// TIA Portal project "FactoryIO_Template_S7-1200_V15_V15.1" (V15.1)
// Vorlageprojekt für das Buch mit Zielsystem S7-1200

(* hardware
DEVICE "S7-1200-Station_1"  S7-1200 Station
   slot 0: "Baugruppenträger_0"  Rack  V1.0
   slot 1: "PLC_1"  CPU 1211C DC/DC/DC  6ES7 211-1AE40-0XB0  V4.1
DEVICE "HMI_1"  KTP900 Basic PN
   slot 0: "HMI_1"  KTP900 Basic PN  6AV2 123-2JB03-0AX0  15.1.0.0
   slot 1: "HMI_RT_1"  KTP900 Basic PN  6AV2 123-2JB03-0AX0  15.1.0.0
   slot 5: "HMI_1.IE_CP_1"  PROFINET Interface  15.0.1.0
      slot 1: "PROFINET Interface_1"  PROFINET Interface
         slot 1: "Port_1"  Port
*)

// ===== PLC "PLC_1"  CPU 1211C DC/DC/DC =====

VAR_GLOBAL   // PLC tag table "Standard-Variablentabelle"
   "Fill valve" AT %A0.0 : Bool;
   "Fill" AT %E0.0 : Bool;
   "Discharge" AT %E0.1 : Bool;
   "Filling" AT %Q0.1 : Bool;
   "Discharge valve" AT %Q0.2 : Bool;
   "Discharging" AT %Q0.3 : Bool;
   "Timer" AT %QD30 : DInt;
   "reset_fill" AT %I0.3 : Bool;
   "reset_empty" AT %I0.4 : Bool;
END_VAR

DATA_BLOCK "Auxiliare"   // DB1
{ S7_Optimized_Access := 'TRUE' }
VERSION : 0.1
   VAR
      timp_setat : Time;
      timp_setat_secunde : Time;
      timp_trecut : Time;
      timp_trecut_secunde_DInt : DInt;
   END_VAR
BEGIN
END_DATA_BLOCK

// folder: System blocks/Program resources

DATA_BLOCK "timer_umplere"   // DB2
{ S7_Optimized_Access := 'TRUE' }
AUTHOR : Simatic
FAMILY : IEC
NAME : IEC_TMR
VERSION : 1.0
// stored: InstanceOfName IEC_TIMER
"IEC_TIMER"
BEGIN
END_DATA_BLOCK

// folder: (top level)

FUNCTION "MHJ-PLC-Lab-Function-S71200" : Void   // FC9000, SCL
{ S7_Optimized_Access := 'TRUE' }
VERSION : 0.1
   VAR_TEMP
      rdTimeReturn : Int;
      outputTime : DTL;
      SyncVal : Byte;
      forVal : Int;
      forVal_2 : Int;
      Value : Byte;
   END_VAR
   VAR CONSTANT
      CompVal : Byte := 16#34;
      Value_01 : Byte := 16#11;
      Value_01_DW : DWord := 16#A165_D992;
      Value_02_DW : DWord := 16#58BE_4401;
   END_VAR
BEGIN

   #Value:=PEEK(area := 16#82,
        dbNumber := 0,
        byteOffset := 511);
   #Value := #Value + 1;

   POKE(area := 16#82,
        dbNumber := 0,
        byteOffset := 511,
        value := #Value);

   POKE(area:=16#81,
        dbNumber:=0,
        byteOffset:=1016,
        value:=#Value_01_DW);
   POKE(area := 16#81,
        dbNumber := 0,
        byteOffset := 1020,
        value := #Value_02_DW);

   POKE(area := 16#81,
        dbNumber := 0,
        byteOffset := 511,
        value := B#16#00);

   FOR #forVal := 0 TO 120 DO
       FOR #forVal_2:=0 TO 10 DO
           #rdTimeReturn:=RD_SYS_T(#outputTime);
           #rdTimeReturn := WR_SYS_T(#outputTime);
           #rdTimeReturn := RD_SYS_T(#outputTime);
           #rdTimeReturn := WR_SYS_T(#outputTime);
       END_FOR;
       #SyncVal:= PEEK(area := 16#81,
                      dbNumber := 0,
                      byteOffset := 511);
       IF #SyncVal = #CompVal THEN
          GOTO M_1;
       END_IF;
   END_FOR;
   RETURN;

   M_1:
   POKE(area := 16#81,
        dbNumber := 0,
        byteOffset := 511,
        value := B#16#0);
END_FUNCTION

ORGANIZATION_BLOCK "Main"   // OB1, LAD, ProgramCycle
TITLE = "Main Program Sweep (Cycle)"
{ S7_Optimized_Access := 'TRUE' }
VERSION : 0.1
   VAR_INPUT
      Initial_Call : Bool;   // Initial call of this OB
      Remanence : Bool;   // =True, if remanent data are available
   END_VAR
BEGIN

REGION Network 1: Konnektierungsbaustein für PLC-Lab
   // Im Netzwerk 1 wird der Konnektierungsbaustein für PLC-Lab aufgerufen.
   // Dieser Aufruf darf nicht entfernt werden!
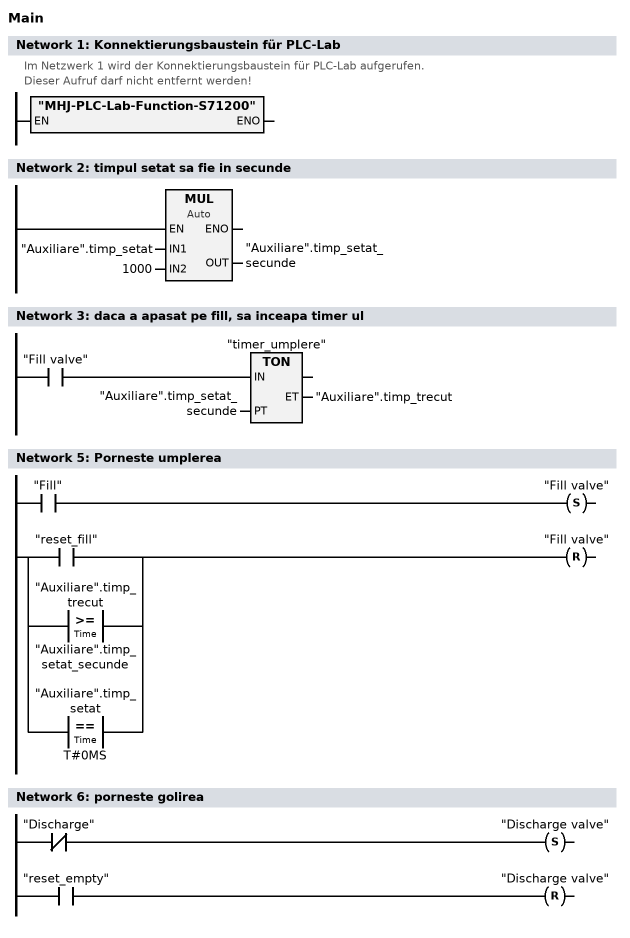
   RUNG wire#powerrail
      "MHJ-PLC-Lab-Function-S71200"()
   END_RUNG
   // the same network as SCL:
   "MHJ-PLC-Lab-Function-S71200"();
END_REGION

REGION Network 2: timpul setat sa fie in secunde
   RUNG wire#powerrail
      Mul(in1 := "Auxiliare".timp_setat, in2 := 1000, out => "Auxiliare".timp_setat_secunde)
   END_RUNG
   // the same network as SCL:
   "Auxiliare".timp_setat_secunde := "Auxiliare".timp_setat * 1000;
END_REGION

REGION Network 3: daca a apasat pe fill, sa inceapa timer ul
   "timer_umplere".TON(IN := "Fill valve", PT := "Auxiliare".timp_setat_secunde, ET => "Auxiliare".timp_trecut);
END_REGION

REGION Network 4 (SCL): timp de afisat in secunde
   "Timer" := TIME_TO_DINT("Auxiliare".timp_trecut / 1000);
END_REGION

REGION Network 5: Porneste umplerea
   RUNG wire#powerrail
      Contact( "Fill" )
      S_Coil( "Fill valve" )
   END_RUNG
   RUNG wire#powerrail
      Contact( "reset_fill" )
      wire#w1
      R_Coil( "Fill valve" )
   END_RUNG
   RUNG wire#powerrail
      { S7_Templates := "SrcType := Time" } GE_Contact(in1 := "Auxiliare".timp_trecut, in2 := "Auxiliare".timp_setat_secunde)
   END_RUNG wire#w1
   RUNG wire#powerrail
      { S7_Templates := "SrcType := Time" } EQ_Contact(in1 := "Auxiliare".timp_setat, in2 := T#0MS)
   END_RUNG wire#w1
   // the same network as SCL:
   IF "Fill" THEN "Fill valve" := TRUE; END_IF;
   IF "reset_fill" OR ("Auxiliare".timp_trecut >= "Auxiliare".timp_setat_secunde) OR ("Auxiliare".timp_setat = T#0MS) THEN
       "Fill valve" := FALSE;
   END_IF;
END_REGION

REGION Network 6: porneste golirea
   RUNG wire#powerrail
      I_Contact( "Discharge" )
      S_Coil( "Discharge valve" )
   END_RUNG
   RUNG wire#powerrail
      Contact( "reset_empty" )
      R_Coil( "Discharge valve" )
   END_RUNG
   // the same network as SCL:
   IF NOT "Discharge" THEN "Discharge valve" := TRUE; END_IF;
   IF "reset_empty" THEN "Discharge valve" := FALSE; END_IF;
END_REGION
END_ORGANIZATION_BLOCK

(* ===== HMI "HMI_RT_1" =====
system functions are stored by id; their names below are inferred from use
connection "HMI_Connection_1": ETHERNET, SMART_S7_1200_OMS

HMI tags "Default tag table"
   "Auxiliare_timp" : Time = PLC Auxiliare.timp_setat, 1 s
   "Auxiliare_timp_trecut_secunde_DInt" : DInt = PLC Auxiliare.timp_trecut_secunde_DInt, 1 s
   "Timer" : DInt = PLC Timer AT %QD30, 1 s
   "Fill" : Bool = PLC Fill AT %I0.0, 1 s
   "Discharge" : Bool = PLC Discharge AT %I0.1, 1 s
   "reset_fill" : Bool = PLC reset_fill AT %I0.3, 1 s
   "reset_empty" : Bool = PLC reset_empty AT %I0.4, 1 s

Template "Template_1" 800x480
   Button "Exit" at 722,440 size 55x39; TextOff 'Exit'; PictureOff "ExitRuntime_KTP900_Basic_PN_TR"; PictureOn "ExitRuntime_KTP900_Basic_PN_TR"
      on Release: StopRuntime(0)
   Button "Template_Button" at 622,440 size 55x39; TextOff 'Text'
   Button "Template_Button_1" at 522,440 size 55x39; TextOff 'Text'
   Button "Template_Button_2" at 422,440 size 55x39; TextOff 'Text'
   Button "Template_Button_3" at 322,440 size 55x39; TextOff 'Text'
   Button "Template_Button_4" at 222,440 size 55x39; TextOff 'Text'
   Button "Template_Button_5" at 122,440 size 55x39; TextOff 'Text'
   Button "Start screen" at 22,440 size 55x39; TextOff 'Start screen'; PictureOff "NavigateHome_KTP900_Basic_PN_TR"; PictureOn "NavigateHome_KTP900_Basic_PN_TR"
      on Release: ActivateScreen("Main", 0)

screen "Main" 800x480, template "Template_1"
   IOField "I/O field_1" at 365,126 size 60x32; FormatPattern 999; Unit s
      ProcessValue <- "Auxiliare_timp"
   TextField "Text field_1" at 357,100 size 74x20; Text 'Timp Setat'
   IOField "I/O field_2" at 366,200 size 59x32; FormatPattern 999; Unit s
      ProcessValue <- "Timer"
   TextField "Text field_2" at 357,176 size 80x20; Text 'Timp Trecut'
   Button "Button_1" at 105,126 size 96x32; TextOff 'Umple'
      on Click: SetBit("Fill")
   Button "Button_2" at 105,196 size 96x32; TextOff 'Reset'
      on Click: SetBit("reset_fill")
   Button "Button_3" at 581,126 size 96x32; TextOff 'Goleste'
      on Click: SetBit("Discharge")
   Button "Button_4" at 581,196 size 96x32; TextOff 'Reset'
      on Click: SetBit("reset_empty")
*)